FUNCTION_BLOCK FB_HandClutchCheck
VAR_INPUT
END_VAR
VAR_OUTPUT
END_VAR
VAR
	m_handClutchSwitch :BOOL;
	m_handClutchOnCounts :INT;
	m_handClutchOnCountThres :INT :=50;
END_VAR

METHOD run : BOOL
VAR_INPUT
	IOValue :UDINT;
END_VAR
// TODO: The two hand clutch switch is mapped to 1/2 bits, but the IO value would change to 28 sometimes
//IF (IOValue AND 10#3) > 0 THEN
IF IOValue > 0 THEN
	m_handClutchOnCounts := MIN(m_handClutchOnCounts +1, m_handClutchOnCountThres);
ELSE
	 m_handClutchOnCounts :=0;
END_IF

m_handClutchSwitch:=m_handClutchOnCounts>=m_handClutchOnCountThres;
run:=m_handClutchSwitch;
END_METHOD

END_FUNCTION_BLOCK

(* stored: Version 1.1.0.1, ProductVersion 3.1.4024.12
   POU FB_HandClutchCheck: Id {2862370c-9cbe-4e26-a065-d84dc0dc8b05}, SpecialFunc None
   Method run: Id {631928bb-17ad-4f7d-bb06-8ffb889b5b39} *)
